# B&R Automation Studio project lab1_MIRTS_save2_4 (part 2)

```iecst
TYPE
    ARNC0FILEMONENTRY_typ : STRUCT
        name                            : UDINT;                                 (* File name (address) *)
        path_name                       : UDINT;                                 (* Full path file name (address) *)
        dir_name                        : UDINT;                                 (* Directory name (address) *)
        device_name                     : UDINT;                                 (* Device name (address) *)
        prog_nr                         : UDINT;                                 (* Number of loaded program *)
        storage_type                    : UDINT;                                 (* Storage type: 1-file, 2-module *)
        time_stamp                      : UDINT;                                 (* File time stamp *)
        precompiled_lcf                 : BOOL;                                  (* Loaded file is laguage configuration file *)
        NOT_USE_1                       : ARRAY[0..2] OF USINT;
        next                            : UDINT;                                 (* Next element in file list *)
    END_STRUCT;
    ARNC0FILEMONBASIC_typ : STRUCT
        name                            : STRING[31];                            (* Name of loaded file *)
        prog_nr                         : UDINT;                                 (* Number of loaded program *)
        storage_type                    : UDINT;                                 (* Storage type: 1-file, 2-module *)
    END_STRUCT;
    ARNC0FILEMONACCESS_typ : STRUCT
        valid                           : BOOL;                                  (* Extended data can be accessed *)
        NOT_USE_1                       : ARRAY[0..2] OF USINT;
        first                           : UDINT;                                 (* Begin of the file list *)
    END_STRUCT;
    ARNC0FILEMON_typ : STRUCT
        set_offset                      : UDINT;                                 (* Required file offset *)
        offset                          : UDINT;                                 (* Offset of displayed files *)
        file                            : ARRAY[0..31] OF ARNC0FILEMONBASIC_typ; (* File monitor *)
        direct_access                   : ARNC0FILEMONACCESS_typ;                (* Access to extended data *)
        handshake                       : BOOL;                                  (* Set to update data *)
        NOT_USE_1                       : ARRAY[0..2] OF USINT;
    END_STRUCT;
    ARNC0EXTWMCOL_typ : STRUCT
        result                          : UDINT;                                 (* WM result *)
        index1                          : UDINT;                                 (* Index of 1st found colliding area *)
        shape1                          : UDINT;                                 (* Shape of colliding area: 1-block, 2-hspace *)
    END_STRUCT;
    ARNC0EXTWM_typ : STRUCT
        joint_position                  : ARRAY[0..11] OF LREAL;                 (* Joint coordinate *)
        xyz_position                    : ARRAY[0..2] OF LREAL;                  (* TCP position if joints cannot be used *)
        D_FULL                          : ARRAY[0..5] OF LREAL;                  (* General tool *)
        local_frame                     : ARRAY[0..5] OF LREAL;                  (* Local (base) frame *)
        collision                       : ARNC0EXTWMCOL_typ;                     (* Additional information about collisions *)
    END_STRUCT;
    OPTMOT_SEG_CONFIG_typ : STRUCT
        distance                        : LREAL;                                 (* Length of the path segments in CNC units *)
        increase_num_seg_from_radius    : LREAL;                                 (* Finer segmentation of circles with smaller radius *)
        increase_num_seg_orient_factor  : LREAL;                                 (* Finer segmentation of orientation change *)
        G126_num_seg                    : UDINT;                                 (* Finer segmentation of rounding edge *)
        G126_num_seg_PTP_Interp         : UDINT;                                 (* Finer segmentation of rounding edge *)
    END_STRUCT;
    OPTMOT_AXES_typ : STRUCT
        ax_count                        : UDINT;                                 (* Number of axes for optimization *)
        ax_index                        : ARRAY [0..14] OF USINT;                (* Index of CNC-axis *)
        NOT_USE_1                       : USINT;
        ax_factor                       : ARRAY [0..14] OF LREAL;                (* Scaling factor *)
    END_STRUCT;
    OPTMOT_PATHDEF_typ : STRUCT
        type                            : UINT;                                  (* Type of path definition *)
        ax_count                        : UINT;                                  (* Number of axes for path computation *)
        ax_index                        : ARRAY [0..14] OF USINT;                (* Index of CNC-axis *)
        NOT_USE_1                       : USINT;
        ax_factor                       : ARRAY [0..14] OF LREAL;                (* Scaling factor *)
    END_STRUCT;
    OPTMOT_TRF_VAR_INSTANCES_typ : STRUCT
        trf_var_ip                      : UDINT;                                 (* For developers only *)
        trf_var_ip_wm                   : UDINT;                                 (* For developers only *)
        trf_var_pp1                     : UDINT;                                 (* For developers only *)
        trf_var_pp2                     : UDINT;                                 (* For developers only *)
        trf_var_bgen                    : UDINT;                                 (* For developers only *)
    END_STRUCT;
    OPTMOT_ACCESS_POINTS_typ : STRUCT
        pp_context                      : UDINT;                                 (* Access of data for external workspace monitoring *)
        wm_function                     : UDINT;                                 (* Access for external call of workspace monitoring *)
        address_debug_data              : UDINT;                                 (* For developers only *)
        trf_var_instances               : OPTMOT_TRF_VAR_INSTANCES_typ;          (* Structure of access points for developers only *)
    END_STRUCT;
    OPTMOT_INTERNAL_typ : STRUCT
        buffer_nc_block                 : UDINT;                                 (* Size of a buffer containing NC-blocks *)
        buffer_geometric_data           : UDINT;                                 (* Size of a buffer containing geometric data of the path *)
        disable_optmot_for_channel      : USINT;                                 (* Deactivation of optimizer for current CNC channel *)
        Ts_multiple                     : USINT;                                 (* Sample time of trajectory planer *)
        linear_feed                     : USINT;                                 (* Behavior of path acceleration *)
        bypass_optmot                   : USINT;                                 (* Simulation mode *)
        addr_dyn_model                  : UDINT;                                 (* Pointer to the dynamic model *)
        der_num_poly_points             : UINT;                                  (* Number of segments used for derivatives computation *)
        geometric_pos_filter            : UINT;                                  (* Number of segments used for position filter *)
        buffer_level_lookahead          : UINT;                                  (* Minimal fill level of lookahead buffer *)
        G220_reduce_to_max_in_buffer    : UINT;                                  (* Reduction of G220 time *)
        sigma_diff_compute              : LREAL;                                 (* Lookahead of segmentation *)
        max_angle                       : LREAL;                                 (* Angle to detect stops on path *)
        access_points                   : OPTMOT_ACCESS_POINTS_typ;              (* Structure of access points for developers only *)
        reserve1                        : ARRAY [0..9] OF LREAL;                 (* For developers only *)
        reserve2                        : ARRAY [0..9] OF DINT;                  (* For developers only *)
    END_STRUCT;
    OPTMOT_LIMITS_typ : STRUCT
        v_joint_min                     : ARRAY [0..14] OF LREAL;                (* Minimal velocity limits of the joint axes *)
        v_joint_max                     : ARRAY [0..14] OF LREAL;                (* Maximal velocity limits of the joint axes *)
        a_joint_min                     : ARRAY [0..14] OF LREAL;                (* Minimal acceleration limits of the joint axes *)
        a_joint_max                     : ARRAY [0..14] OF LREAL;                (* Maximal acceleration limits of the joint axes *)
        j_joint_min                     : ARRAY [0..14] OF LREAL;                (* Minimal jerk limits of the joint axes *)
        j_joint_max                     : ARRAY [0..14] OF LREAL;                (* Maximal jerk limits of the joint axes *)
        torque_min                      : ARRAY [0..14] OF LREAL;                (* Minimal torque limits of the joint axes *)
        torque_max                      : ARRAY [0..14] OF LREAL;                (* Maximal torque limits of the joint axes *)
        torque_limits_in_generator_mode : UDINT;                                 (* Activation of generator mode *)
        torque_gen_factor_min           : ARRAY [0..14] OF LREAL;                (* Factor for minimal torque limit in generator mode *)
        torque_gen_factor_max           : ARRAY [0..14] OF LREAL;                (* Factor for maximal torque limit in generator mode *)
        v_path_min                      : ARRAY [0..31] OF LREAL;                (* Minimal velocity limits of the path definitions *)
        v_path_max                      : ARRAY [0..31] OF LREAL;                (* Maximal velocity limits of the path definitions *)
        a_path_min                      : ARRAY [0..31] OF LREAL;                (* Minimal acceleration limits of the path definitions *)
        a_path_max                      : ARRAY [0..31] OF LREAL;                (* Maximal acceleration limits of the path definitions *)
        j_path_min                      : ARRAY [0..31] OF LREAL;                (* Minimal jerk limits of the path definitions *)
        j_path_max                      : ARRAY [0..31] OF LREAL;                (* Maximal jerk limits of the path definitions *)
    END_STRUCT;
    OPTMOT_ACTIVE_LIMIT_typ : STRUCT
        type                            : USINT;                                 (* Type of the active limit *)
        source                          : USINT;                                 (* Source of the active limit *)
        min_max                         : SINT;                                  (* Positive or negative range of the active limit *)
        index                           : USINT;                                 (* Index of the axis or path definition of the active limit *)
    END_STRUCT;
    OPTMOT_UNFILTERED_MONITOR_typ : STRUCT
        s_joint                         : ARRAY [0..14] OF LREAL;                (* Cyclical joint position in CNC units *)
        v_joint                         : ARRAY [0..14] OF LREAL;                (* Cyclical joint velocity in CNC units *)
        a_joint                         : ARRAY [0..14] OF LREAL;                (* Cyclical joint acceleration in CNC units *)
        j_joint                         : ARRAY [0..14] OF LREAL;                (* Cyclical joint jerk in CNC units *)
    END_STRUCT;
    OPTMOT_MONITOR_typ : STRUCT
        s_joint                         : ARRAY [0..14] OF LREAL;                (* Cyclical joint position in CNC units *)
        v_joint                         : ARRAY [0..14] OF LREAL;                (* Cyclical joint velocity in CNC units *)
        a_joint                         : ARRAY [0..14] OF LREAL;                (* Cyclical joint acceleration in CNC units *)
        j_joint                         : ARRAY [0..14] OF LREAL;                (* Cyclical joint jerk in CNC units *)
        feed_forward_torque             : ARRAY [0..14] OF LREAL;                (* Cyclical joint torque/force *)
        v_path                          : ARRAY [0..31] OF LREAL;                (* Cyclical path velocity in CNC units *)
        unfiltered_monitor              : OPTMOT_UNFILTERED_MONITOR_typ;         (* Monitor data without filters and override *)
        active_limit                    : OPTMOT_ACTIVE_LIMIT_typ;               (* Structure of information about current limitation *)
        data_valid                      : UINT;                                  (* Feed forward data is valid *)
        fill_level_lookahead            : UINT;                                  (* Fill level of lookahead buffer *)
        reserve                         : ARRAY [0..1] OF UDINT;
    END_STRUCT;
    OPTMOT_COND_STOP_typ : STRUCT
        active                          : UINT;                                  (* Conditional stop active *)
        call_stop_internal              : UINT;                                  (* Internal execution of the conditional stop *)
        identifier                      : UDINT;                                 (* Identifier of the conditional stop *)
        select_overlapped_identifier    : UDINT;                                 (* Selection of identifier in overlapping conditional stops *)
        select_identifier_stop_internal : UDINT;                                 (* Selection of identifier if conditional stop is executed internally *)
    END_STRUCT;
    OPTMOT_COND_STOP_OPTMOT_typ : STRUCT
        identifier_aktiv                : UDINT;                                 (* Output of aktive identifier *)
        identifier_fulfilled            : UDINT;                                 (* Input of fulfilled identifier *)
    END_STRUCT;
    OPTMOT_STOPPING_typ : STRUCT
        G126_skip_if_stop               : UINT;                                  (* Skip G126 if a stop on path occurs *)
        trajectory                      : UINT;                                  (* Definition of stopping trajectory *)
        conditional_stop                : OPTMOT_COND_STOP_typ;                  (* Structure of conditional stop *)
        conditional_stop_optmot         : OPTMOT_COND_STOP_OPTMOT_typ;           (* Structure of optmot synchronal conditional stop *)
    END_STRUCT;
    OPTMOT_PATH_typ : STRUCT
        G126_skip_smaller_radius        : LREAL;                                 (* Skip G126 if programmed radius is smaller *)
        G126_round_whole_line           : UDINT;                                 (* Round whole first/last line *)
        count                           : UDINT;                                 (* Number of path definitions *)
        definition                      : ARRAY [0..31] OF OPTMOT_PATHDEF_typ;   (* Structure of path definitions parameters *)
        stopping                        : OPTMOT_STOPPING_typ;                   (* Structure of stopping parameters *)
        reserve1                        : ARRAY [0..170] OF UDINT;
    END_STRUCT;
    OPTMOT_CONFIG_typ : STRUCT
        axes                            : OPTMOT_AXES_typ;                       (* Structure of joint axes parameters *)
        path                            : OPTMOT_PATH_typ;                       (* Structure of path parameters *)
        limits                          : ARRAY [0..31] OF OPTMOT_LIMITS_typ;    (* Structure of limit parameters *)
        segmentation                    : OPTMOT_SEG_CONFIG_typ;                 (* Structure of segmentation parameters *)
        monitor                         : OPTMOT_MONITOR_typ;                    (* Structure of monitor parameters *)
        internals                       : OPTMOT_INTERNAL_typ;                   (* Structure of internal parameters *)
    END_STRUCT;
    OPTMOT_MONITOR_ADVANCED_typ : STRUCT
        s_joint                         : ARRAY [0..14] OF LREAL;                (* Cyclical joint position in CNC units *)
        v_joint                         : ARRAY [0..14] OF LREAL;                (* Cyclical joint velocity in CNC units *)
        a_joint                         : ARRAY [0..14] OF LREAL;                (* Cyclical joint acceleration in CNC units *)
        j_joint                         : ARRAY [0..14] OF LREAL;                (* Cyclical joint jerk in CNC units *)
        feed_forward_torque             : ARRAY [0..14] OF LREAL;                (* Cyclical joint torque/force *)
        v_path                          : ARRAY [0..31] OF LREAL;                (* Cyclical path velocity in CNC units *)
        unfiltered_monitor              : OPTMOT_UNFILTERED_MONITOR_typ;         (* Monitor data without filters and override *)
        active_limit                    : OPTMOT_ACTIVE_LIMIT_typ;               (* Structure of information about current limitation *)
        data_valid                      : UINT;                                  (* Feed forward data is valid *)
        fill_level_lookahead            : UINT;                                  (* Fill level of lookahead buffer *)
        tracking_active                 : UINT;                                  (* Tracking active *)
        tracking_synch                  : UINT;                                  (* Robot synchronized with conveyor *)
        tracking_index                  : UINT;                                  (* Active tracking index *)
        reserve                         : UINT;
    END_STRUCT;
    OPTMOT_TRACKING_ORIENTATION_typ : STRUCT
        phi                             : LREAL;                                 (* Phi-component of a rotation *)
        theta                           : LREAL;                                 (* Theta-component of a rotation *)
        psi                             : LREAL;                                 (* Psi-component of a rotation *)
    END_STRUCT;
    OPTMOT_TRACKING_ORIENT_PARAM_typ : STRUCT
        measure                         : UDINT;                                 (* Unit of measurement of the angles *)
        angles_type                     : UDINT;                                 (* Angles type *)
    END_STRUCT;
    OPTMOT_TRACKING_LIMITS_typ : STRUCT
        maxVelocity                     : LREAL;                                 (* Maximal velocity of the conveyor belt *)
    END_STRUCT;
    OPTMOT_TRACKING_CYCLIC_typ : STRUCT
        position                        : LREAL;                                 (* Cyclical position of the conveyor belt *)
        velocity                        : LREAL;                                 (* Cyclical velocity of the conveyor belt *)
    END_STRUCT;
    OPTMOT_TRACKING_CONVEYOR_typ : STRUCT
        limits                          : OPTMOT_TRACKING_LIMITS_typ;            (* Structure of conveyor limits *)
        orientation                     : OPTMOT_TRACKING_ORIENTATION_typ;       (* Structure of orientation between global basic frame and conveyor belt frame *)
        cyclicData                      : OPTMOT_TRACKING_CYCLIC_typ;            (* Structure of cyclic data *)
    END_STRUCT;
    OPTMOT_TRACKING_CONVEYORDATA_typ : STRUCT
        orientationParameter            : OPTMOT_TRACKING_ORIENT_PARAM_typ;      (* Structure of general orientation parameters *)
        conveyor                        : ARRAY [0..9] OF OPTMOT_TRACKING_CONVEYOR_typ; (* Structure of conveyor belt data *)
    END_STRUCT;
    OPTMOT_TRACKING_typ : STRUCT
        enable                          : UDINT;                                 (* Enable tracking *)
        conveyorData                    : OPTMOT_TRACKING_CONVEYORDATA_typ;      (* Structure of conveyor belt tracking *)
        reserve1                        : ARRAY [0..7] OF LREAL;                 (* For developers only *)
        reserve2                        : ARRAY [0..31] OF UDINT;                (* For developers only *)
    END_STRUCT;
    OPTMOT_PATH_ADVANCED_typ : STRUCT
        G126_skip_smaller_radius        : LREAL;                                 (* Skip G126 if programmed radius is smaller *)
        G126_round_whole_line           : UDINT;                                 (* Round whole first/last line *)
        count                           : UDINT;                                 (* Number of path definitions *)
        definition                      : ARRAY [0..31] OF OPTMOT_PATHDEF_typ;   (* Structure of path definitions parameters *)
        stopping                        : OPTMOT_STOPPING_typ;                   (* Structure of stopping parameters *)
        tracking                        : OPTMOT_TRACKING_typ;                   (* Structure of tracking parameters *)
    END_STRUCT;
    OPTMOT_CONFIG_ADVANCED_typ : STRUCT
        axes                            : OPTMOT_AXES_typ;                       (* Structure of joint axes parameters *)
        path                            : OPTMOT_PATH_ADVANCED_typ;              (* Structure of path parameters *)
        limits                          : ARRAY [0..31] OF OPTMOT_LIMITS_typ;    (* Structure of limit parameters *)
        segmentation                    : OPTMOT_SEG_CONFIG_typ;                 (* Structure of segmentation parameters *)
        monitor                         : OPTMOT_MONITOR_ADVANCED_typ;           (* Structure of monitor parameters *)
        internals                       : OPTMOT_INTERNAL_typ;                   (* Structure of internal parameters *)
    END_STRUCT;
    ARNC0PLOTDATA01_typ : STRUCT
        block_ncprog                    : UDINT;                       			 (* Block number *)
        line_ncprog                     : UDINT;                       			 (* Line number *)
        MpId                            : UDINT;                       			 (* Motion packet ident *)
        MpSubId                         : UDINT;                       			 (* Motion packet subident *)
        cmd_code                        : UINT;                       			 (* Command *)
        reserve                         : UINT;                       			 (* don't use *)
        data                            : ARRAY [0..51] OF USINT;                (* Data *)
    END_STRUCT;
    ARNC0PLOTDATA02_typ : STRUCT
        block_ncprog                    : UDINT;                       			 (* Block number *)
        line_ncprog                     : UDINT;                       			 (* Line number *)
        MpId                            : UDINT;                       			 (* Motion packet ident *)
        MpSubId                         : UDINT;                       			 (* Motion packet subident *)
        cmd_code                        : UINT;                       			 (* Command *)
        reserve                         : UINT;                       			 (* don't use *)
        data                            : ARRAY [0..51] OF USINT;                (* Data *)
    END_STRUCT;
    ARNC0PLDMOVE_typ : STRUCT
        ep                              : ARRAY [0..2] OF REAL;                  (* End point *)
        cp                              : ARRAY [0..2] OF REAL;                  (* Center point *)
        radius                          : REAL;                                  (* Tool radius *)
        v_ncprog                        : REAL;                                  (* Programmed feedrate *)
        info                            : UDINT;                                 (* Info bits *)
    END_STRUCT;
    ARNC0PLDMOVE02_typ : STRUCT
        ep                              : ARRAY [0..2] OF REAL;                  (* End point *)
        cp                              : ARRAY [0..2] OF REAL;                  (* Center point *)
        radius                          : REAL;                                  (* Tool radius *)
        v_ncprog                        : REAL;                                  (* Programmed feedrate *)
        t                               : REAL;                                  (* block runtime *)
        s                               : REAL;                                  (* block length, interpolated axes *)
        s_all                           : REAL;                                  (* block length, all axes *)
        info                            : UDINT;                                 (* Info bits *)
    END_STRUCT;
    ARNC0PLDPROGEND_typ : STRUCT
        t                               : REAL;                                  (* estimated runtime *)
        s                               : REAL;                                  (* path length, interpolated axes *)
        s_all                           : REAL;                                  (* path length, all axes *)
    END_STRUCT;
    ARNC0PLDPROGSTART_typ : STRUCT
        ProgNumber                      : UDINT;                                 (* program number *)
    END_STRUCT;
    ARNC0PLDTOOL_typ : STRUCT
        radius                          : REAL;                                  (* Tool radius *)
        length                          : REAL;                                  (* Tool length *)
        offset                          : ARRAY [0..2] OF REAL;                  (* Tool offset *)
        index                           : UINT;                                  (* Tool index, tool data number *)
        reserve                         : UINT;                                  (* don't use *)
    END_STRUCT;
    ARNC0PLDCSTRF_typ : STRUCT
        matrix                          : ARRAY [0..8] OF REAL;                  (* Rotation matrix *)
        offset                          : ARRAY [0..2] OF REAL;                  (* Offset (cs + tool) *)
        info                            : UDINT;                                 (* Info bits *)
    END_STRUCT;
    ARNC0PLDUSER_typ : STRUCT
        data                            : ARRAY [0..51] OF USINT;                (* User data *)
    END_STRUCT;
    ARNC0TRFIODATA_typ : STRUCT
        status                          : UDINT;                                 (* Return status of the last call of the transformation function *)
        in_pos                          : ARRAY [0..11] OF LREAL;                (* Input positions of the transformation function *)
        in_pos_ext                      : ARRAY [0..11] OF LREAL;                (* Extended input positions of the transformation function *)
        out_pos                         : ARRAY [0..71] OF LREAL;                (* Output positions of the transformation function *)
        info                            : ARRAY [0..8] OF UDINT;                 (* Information about the last call of the transformation function *)
    END_STRUCT;
    ARNC0WSCTRL_typ : STRUCT
        link_index                      : UDINT;                                 (* index of colliding link *)
        link2_index                     : UDINT;                                 (* index of colliding link for self-collision *)
        area_index                      : UDINT;                                 (* index of colliding area *)
    END_STRUCT;
    ARNC0NCMON_EXT_AX_typ : STRUCT
        nc_object                       : UDINT;
        nc_object_plcopen               : UDINT;
        v                               : REAL;                                  (* axis limit [cnc unit/s] *)
        a                               : REAL;                                  (* axis limit [cnc unit/s2] *)
        t_jolt                          : REAL;                                  (* axis jolt filter [s] (cnc system) *)
        pos_sw_end                      : DINT;                                  (* [cnc unit] *)
        neg_sw_end                      : DINT;                                  (* [cnc unit] *)
        unitfactor                      : REAL;                                  (* cnc unit factor *)
        plcopen_factor                  : REAL;                                  (* PLCopen unit factor *)
        type                            : UDINT;                                 (* axis type *)
        rot_period                      : REAL;                                  (* period of the rotary axis [cnc unit] *)
        rot_offset                      : REAL;                                  (* period start offsetof the rotary axis [cnc unit] *)
        ipl_mode                        : USINT;                                 (* interpolation mode *)
        drive_axfilter                  : USINT;                                 (* axis jolt filter on drive enable/disable *)
        nc_obj_name                     : ARRAY [0..13] OF USINT;
        cnc_ax_name                     : ARRAY [0..13] OF USINT;
        reserve                         : ARRAY [0..1] OF USINT;
    END_STRUCT;
    ARNC0NCMON_EXT_G113_typ : STRUCT
        k_alpha_max                     : REAL;                                  (* G113 parameter *)
        alpha_min                       : REAL;                                  (* G113 parameter *)
        alpha_max                       : REAL;                                  (* G113 parameter *)
    END_STRUCT;
    ARNC0NCMON_EXT_CNC_typ : STRUCT
        nc_object                       : UDINT;                                 (* nc object (cnc) *)
        v                               : REAL;                                  (* path limit [cnc unit/s] *)
        a_pos                           : REAL;                                  (* path limit [cnc unit/s2] *)
        a_neg                           : REAL;                                  (* path limit [cnc unit/s] *)
        t_jolt                          : REAL;                                  (* path jolt filter [s] *)
        feed                            : REAL;                                  (* programmed feed [cnc unit/s] *)
        v_jump                          : ARRAY [0..14] OF REAL;                 (* speed jump [cnc unit/s] *)
        a_jump                          : ARRAY [0..14] OF REAL;                 (* acceleration jump [cnc unit/s] *)
        v_jump_t                        : REAL;                                  (* speed jump for tangential axes [cnc unit/s] *)
        s_jump_t                        : REAL;                                  (* blocktransition tangential / non tangential [deg] *)
        filter_err_cir                  : REAL;                                  (* allowed radius error (jolt filter) [cnc unit] *)
        filter_err_trans                : REAL;                                  (* contour violation (jolt filter) [cnc unit] *)
        radius_err                      : REAL;                                  (* center point prgramming [cnc unit] *)
        elements                        : UDINT;                                 (* calculated elements before start *)
        block_buffer                    : UDINT;                                 (* block buffer for backtracing *)
        lookahead                       : UDINT;                                 (* look ahead buffer (dynamics calculation) *)
        first_M                         : UINT;                                  (* index of 1st M function (without sync) *)
        last_M                          : UINT;                                  (* index of last M function (without sync) *)
        first_M_S                       : UINT;                                  (* index of 1st M function (with sync) *)
        last_M_S                        : UINT;                                  (* index of last M function (with sync) *)
        s_sync1_t                       : UINT;                                  (* 1st sync M function (G141) *)
        s_sync2_t                       : UINT;                                  (* 2nd sync M function (G141) *)
        blocktransition                 : USINT;                                 (* block transition mode *)
        reserve                         : USINT;
        nc_obj_name                     : ARRAY [0..13] OF USINT;
        g113_data                       : ARNC0NCMON_EXT_G113_typ;
    END_STRUCT;
    ARNC0NCMON_EXT_G705_typ : STRUCT
        ident                           : UDINT;                                 (* G705 ident *)
        axis                            : ARRAY[0..14] OF ARNC0NCMON_EXT_AX_typ;
        cnc                             : ARNC0NCMON_EXT_CNC_typ;
        block_ncprog                    : UDINT;                                 (* block number (G705) *)
        line_ncprog                     : UDINT;                                 (* line number (G705) *)
        cnc_channel                     : UINT;                                  (* cnc channel (idndex) *)
        reserve                         : UINT;
    END_STRUCT;
    ARNC0NCMON_EXT_typ : STRUCT
        s_set                           : ARRAY [0..14] OF LREAL;                (* set position *)
        s_ncprog                        : LREAL;                                 (* path position in current CNC program *)
        g705_data                       : ARNC0NCMON_EXT_G705_typ;               (* parameter at program start, at G705 *)
        reserve                         : ARRAY[0..1] OF UDINT;
    END_STRUCT;
    ARNC0WFM_SERIAL_typ : STRUCT
        nr_of_points : UDINT;                                                    (* number of points of wire-frame model *)
        point : ARRAY[0..20, 0..2] OF LREAL;                                     (* points of wire-frame model *)
        nr_of_arms : UDINT;                                                      (* number of arm diameters *)
        arm_diameter : ARRAY[0..19] OF LREAL;                                    (* arm diameters *)
        safe_distance : LREAL;                                                   (* safe distance *)
    END_STRUCT;
    ARNC0WFM_COMPLETE_typ : STRUCT
        data : ARRAY[0..329] OF UDINT;                                           (* internal data of complete wire-frame model *)
    END_STRUCT;
    ARNC0WFM_typ : STRUCT
        use_complete : UDINT;                                                    (* use complete type of wire-frame model *)
        complete : ARNC0WFM_COMPLETE_typ;                                        (* complete wire-frame model data *)
        use_serial : UDINT;                                                      (* use serial type of wire-frame model *)
        serial : ARNC0WFM_SERIAL_typ;                                            (* serial wire-frame model data *)
    END_STRUCT;
    ARNC0WFM_BFS : STRUCT
        enable : UDINT;                                                          (* enable frame *)
        dx : LREAL;                                                              (* x transition *)
        dy : LREAL;                                                              (* y transition *)
        dz : LREAL;                                                              (* z transition *)
        phi : LREAL;                                                             (* angle in meaning of angles type *)
        theta : LREAL;                                                           (* angle in meaning of angles type *)
        psi : LREAL;                                                             (* angle in meaning of angles type *)
        angles_type : UDINT;                                                     (* angles type *)
    END_STRUCT;
    ARNC0WFM_MON_typ : STRUCT
        valid_data : UDINT;                                                      (* number of calls with valid data *)
        invalid_data : UDINT;                                                    (* number of calls with invalid data *)
    END_STRUCT;
    ARNC0WFM_EXT_typ : STRUCT
        p_wire_frame_model : REFERENCE TO ARNC0WFM_typ;                          (* reference to wire-frame model data *)
        base_frame_shift : ARNC0WFM_BFS;                                         (* frame *)
        monitor : ARNC0WFM_MON_typ;                                              (* monitor *)
    END_STRUCT;
    ARNC0INTERACTION_typ : STRUCT
        wire_frame_model : ARNC0WFM_typ;                                         (* wire-frame model data *)
        wire_frame_models_to_check : ARRAY[0..23]OF ARNC0WFM_EXT_typ;            (* array of wire-frame models data *)
    END_STRUCT;
END_TYPE
TYPE
  ARNC0IP_MON_typ : STRUCT
    enable : USINT;                             (*Enable cyclic update *)
    reserve : ARRAY[0..2] OF USINT;             (*[RESERVE] *)
    status_msg : ARRAY[0..79] OF USINT;         (*String: current status of interpreter e.g. Running/Waiting/Finished *)
    last_error_msg : ARRAY[0..119] OF USINT;    (*String: last error message issued *)
    last_error_code : UINT ;                    (*Last status message code issued *)
    loaded_prog_count : UINT ;                  (*Number of files loaded *)
    prog_name : ARRAY[0..79] OF USINT;          (*Name of start-program *)
    ncblock_l2 : ARRAY[0..79] OF USINT;         (*Interpeter block monitor: current line -2 *)
    ncblock_l1 : ARRAY[0..79] OF USINT;         (*Interpeter block monitor: current line -1 *)
    ncblock : ARRAY[0..79] OF USINT;            (*Interpeter block monitor: current line *)
    ncblock_n1 : ARRAY[0..79] OF USINT;         (*Interpeter block monitor: current line +1 *)
    ncblock_n2 : ARRAY[0..79] OF USINT;         (*Interpeter block monitor: current line +2 *)
    cur_line_num : UDINT ;                      (*Interpeter block monitor: current line number *)
    cur_block_num : UDINT ;                     (*Interpeter block monitor: current line N-block number *)
    intern1 : UDINT ;                           (*[INTERNAL] *)
    intern2 : UDINT ;                           (*[INTERNAL] *)
    intern3 : UDINT ;                           (*[INTERNAL] *)
    intern4 : UDINT ;                           (*[INTERNAL] *)
    intern5 : UDINT ;                           (*[INTERNAL] *)
    breakpoint_count : UDINT ;                  (*Number of breakpoints set *)
    ipvar_access_count : UDINT ;                (*Number of IP variables being directly accessed by PLC *)
    intern6 : UDINT ;                           (*[INTERNAL] *)
    intern7 : UDINT ;                           (*[INTERNAL] *)
    num_parallel_events : UDINT ;               (*Number of cyclic jobs currently active *)
    parallel_cycle_count : UDINT ;              (*Number of execution cycles of all cyclic jobs *)
    parallel_action_text : ARRAY[0..11, 0..79] OF USINT; (*cyclic execution monitor - cyclic job source line text *)
    parallel_eval_count : ARRAY[0..11] OF UDINT ;   (*number of times the cyclic job has been evaluated (tested) *)
    parallel_exec_count : ARRAY[0..11] OF UDINT ;   (*number of times a Synchronised Action has executed (not relevant to FUBs) *)
    num_fubs_exec_ipsynch : UDINT ;             (*Number of interpreter synchronous FUBs executing *)
    num_fubs_exec_ppsynch : UDINT ;             (*Number of path synchronous FUBs executing *)
    callstack : ARRAY[0..11, 0..79] OF USINT;   (*Program callstack *)
    shared_mem_size : UDINT ;                   (*Memory consumed by shared library data (partitions will be larger) *)
    ip_mem_size : UDINT ;                       (*Memory consumed by interpreter instance (partitions will be larger) *)
    ip_cur_file_mem_size : UDINT ;              (*Memory consumed by start program (or last loaded program) file (partitions will be larger) *)
    sys_free_mem : UDINT ;                      (*Available system memory *)
    intern8 : UDINT ;                           (*[INTERNAL] *)
    intern9 : UDINT ;                           (*[INTERNAL] *)
    intern10 : UDINT ;                          (*[INTERNAL] *)
    intern11 : UDINT ;                          (*[INTERNAL] *)
    parallel_enabled : USINT ;                  (*Bool: cyclic execution enabled *)
    parallel_rdisable_set : USINT ;             (*Bool: cyclic jobs set the keep-alive (rdisable) flag *)
    intern12 : USINT ;                          (*[INTERNAL] *)
    intern13 : USINT ;                          (*[INTERNAL] *)
    cur_prog_file_name : ARRAY[0..79] OF USINT ;(*File name of the current program*)
    cur_prog_name : ARRAY[0..79] OF USINT ;     (*Name of the current program*)
  END_STRUCT;
END_TYPE
```

- acp10err-en.txt (not shown)

- arnc0err-de.txt (not shown)

- arnc0err-en.txt (not shown)

### Library Logical/Libraries/MotorCntrl (ANSIC)

#### MotorCntrl.fun - Exported functions and function blocks
```iecst
{REDUND_ERROR} FUNCTION_BLOCK FB_Motor (*TODO: Add your comment here*) (*$GROUP=User,$CAT=User,$GROUPICON=User.png,$CATICON=User.png*)
	VAR_INPUT
		u : {REDUND_UNREPLICABLE} REAL; (*Входное напряжение [B]*)
	END_VAR
	VAR_OUTPUT
		w : REAL; (*Частота вращения [об/мин]*)
		phi : REAL; (*Положение [рад]*)
	END_VAR
	VAR
		integrator : FB_Integrator; (*Интегратор*)
		Tm : REAL; (*Электромеханическая постоянная времени [с]*)
		ke : REAL; (*Постоянная ЭДС двигателя [В*мин/об]*)
		dt : REAL; (*Шаг расчета [с]*)
	END_VAR
END_FUNCTION_BLOCK

{REDUND_ERROR} FUNCTION_BLOCK FB_Regulator (*TODO: Add your comment here*) (*$GROUP=User,$CAT=User,$GROUPICON=User.png,$CATICON=User.png*)
	VAR_INPUT
		e : {REDUND_UNREPLICABLE} REAL; (*Рассогласование между задающим воздействием и реальной скоростью вращения вала ДПТ [об/мин]*)
	END_VAR
	VAR_OUTPUT
		u : REAL; (*Напряжение, подаваемое на вход ДПТ [B]*)
	END_VAR
	VAR
		k_p : REAL; (*Пропорциональный коэффициент регулятора*)
		k_i : REAL; (*Интегральный коэффициент регулятора*)
		integrator : FB_Integrator; (*Интегратор*)
		ivOld : REAL; (*Хранение предыдущего значения схемы противонакопления*)
		max_abs_value : REAL; (*Граница блока ограничения [В]*)
		dt : REAL; (*Шаг расчета [c]*)
	END_VAR
END_FUNCTION_BLOCK

{REDUND_ERROR} FUNCTION_BLOCK FB_Integrator (*TODO: Add your comment here*) (*$GROUP=User,$CAT=User,$GROUPICON=User.png,$CATICON=User.png*)
	VAR_INPUT
		in : {REDUND_UNREPLICABLE} REAL; (*Вход интегрирующего звена*)
	END_VAR
	VAR_OUTPUT
		out : REAL; (*Выход интегрирующего звена*)
	END_VAR
	VAR
		dt : REAL; (*Шаг расчета [c]*)
	END_VAR
END_FUNCTION_BLOCK
```

#### FB_Motor.c
```c
#include <bur/plctypes.h>
#ifdef __cplusplus
	extern "C"
	{
#endif
#include "MotorCntrl.h"
#ifdef __cplusplus
	};
#endif
/* TODO: Add your comment here */
void FB_Motor(struct FB_Motor* inst)
{
	/*TODO: Add your code here*/
	inst->integrator.dt = inst->dt;
	inst->integrator.in = ((inst->u)/(inst->ke) - (inst->w))*\
		(1/(inst->Tm));
	FB_Integrator(&(inst->integrator));
	inst->w = inst->integrator.out;
	inst->integrator.in = inst->w;
	inst->integrator.out = inst->phi;
	FB_Integrator(&(inst->integrator));
	inst->phi = inst->integrator.out;
	inst->integrator.out = inst->w;
}
```

#### FB_Regulator.c
```c
#include <bur/plctypes.h>
#ifdef __cplusplus
	extern "C"
	{
#endif
#include "MotorCntrl.h"
#ifdef __cplusplus
	};
#endif
/* TODO: Add your comment here */
REAL V_lim(REAL in, REAL max_in)
{
	if ((in >= max_in) || (in <= -max_in))
	{
		if (in>0)
			return max_in;
		else
			return -max_in;
	}
	else
		return in;
}
void FB_Regulator(struct FB_Regulator* inst)
{
	/*TODO: Add your code here*/
	REAL temp;
	inst->integrator.dt = inst->dt;
	inst->integrator.in = ((inst->e*inst->k_i)+inst->ivOld);
	FB_Integrator(&(inst->integrator));
	temp = inst->integrator.out + V_lim((inst->e)*(inst->k_p),inst->max_abs_value);
	inst->u = V_lim(temp, inst->max_abs_value);
	inst->ivOld = inst->u - temp;
}
```

#### FB_Integrator.c
```c
#include <bur/plctypes.h>
#ifdef __cplusplus
	extern "C"
	{
#endif
#include "MotorCntrl.h"
#ifdef __cplusplus
	};
#endif
/* TODO: Add your comment here */
void FB_Integrator(struct FB_Integrator* inst)
{
	/*TODO: Add your code here*/
	inst->out += (inst->in)*(inst->dt);
}
```

### Program Logical/LedCtrl (ANSIC)

#### Main.c
```c
#include <bur/plctypes.h>

#ifdef _DEFAULT_INCLUDES
	#include <AsDefault.h>
#endif

void _INIT ProgramInit(void)
{

}

void _CYCLIC ProgramCyclic(void)
{
		sc0 = sw0;
		sc1 = sw1;
		sc2 = sw2;
		sc3 = sw3;

}

void _EXIT ProgramExit(void)
{

}
```

### Program Logical/ncsdcctrl

#### ncsdcctrl.var
```iecst
VAR
	gAxis01_oSetPosOld : INT := 0;
	gAxis02_oSetPosOld : INT := 0;
	gAxis04_oSetPosOld : INT := 0;
	gAxis05_oSetPosOld : INT := 0;
END_VAR
```

#### ncsdcctrlCyclic.st
```iecst
PROGRAM _CYCLIC

(* ### BEGIN gAxis01 ### *)

(* life counter emulation of digital inputs *)
      gAxis01_DiDoIf.iLifeCntReference := gAxis01_DiDoIf.iLifeCntReference + 1;
      gAxis01_DiDoIf.iLifeCntNegHwEnd  := gAxis01_DiDoIf.iLifeCntNegHwEnd  + 1;
      gAxis01_DiDoIf.iLifeCntPosHwEnd  := gAxis01_DiDoIf.iLifeCntPosHwEnd  + 1;

(* default function model of ACOPOSmicro: convert absolute steps to delta steps - overflow save delta calculation *)
      gAxis01_MotorStep0 := gAxis01_DrvIf.oSetPos - gAxis01_oSetPosOld;
      gAxis01_oSetPosOld := gAxis01_DrvIf.oSetPos;

(* ### END gAxis01 ### *)

(* ### BEGIN gAxis02 ### *)

(* life counter emulation of digital inputs *)
      gAxis02_DiDoIf.iLifeCntReference := gAxis02_DiDoIf.iLifeCntReference + 1;
      gAxis02_DiDoIf.iLifeCntNegHwEnd  := gAxis02_DiDoIf.iLifeCntNegHwEnd  + 1;
      gAxis02_DiDoIf.iLifeCntPosHwEnd  := gAxis02_DiDoIf.iLifeCntPosHwEnd  + 1;

(* default function model of ACOPOSmicro: convert absolute steps to delta steps - overflow save delta calculation *)
      gAxis02_MotorStep0 := gAxis02_DrvIf.oSetPos - gAxis02_oSetPosOld;
      gAxis02_oSetPosOld := gAxis02_DrvIf.oSetPos;

(* ### END gAxis02 ### *)

(* ### BEGIN gAxis03 ### *)

(* life counter emulation of digital inputs *)
        gAxis03_DiDoIf.iLifeCntReference := gAxis03_DiDoIf.iLifeCntReference + 1;
        gAxis03_DiDoIf.iLifeCntNegHwEnd  := gAxis03_DiDoIf.iLifeCntNegHwEnd  + 1;
        gAxis03_DiDoIf.iLifeCntPosHwEnd  := gAxis03_DiDoIf.iLifeCntPosHwEnd  + 1;

(* ### END gAxis03 ### *)

(* ### BEGIN gAxis04 ### *)

(* life counter emulation of digital inputs *)
      gAxis04_DiDoIf.iLifeCntReference := gAxis04_DiDoIf.iLifeCntReference + 1;
      gAxis04_DiDoIf.iLifeCntNegHwEnd  := gAxis04_DiDoIf.iLifeCntNegHwEnd  + 1;
      gAxis04_DiDoIf.iLifeCntPosHwEnd  := gAxis04_DiDoIf.iLifeCntPosHwEnd  + 1;

(* default function model of ACOPOSmicro: convert absolute steps to delta steps - overflow save delta calculation *)
      gAxis04_MotorStep0 := gAxis04_DrvIf.oSetPos - gAxis04_oSetPosOld;
      gAxis04_oSetPosOld := gAxis04_DrvIf.oSetPos;

(* ### END gAxis04 ### *)

(* ### BEGIN gAxis05 ### *)

(* life counter emulation of digital inputs *)
      gAxis05_DiDoIf.iLifeCntReference := gAxis05_DiDoIf.iLifeCntReference + 1;
      gAxis05_DiDoIf.iLifeCntNegHwEnd  := gAxis05_DiDoIf.iLifeCntNegHwEnd  + 1;
      gAxis05_DiDoIf.iLifeCntPosHwEnd  := gAxis05_DiDoIf.iLifeCntPosHwEnd  + 1;

(* default function model of ACOPOSmicro: convert absolute steps to delta steps - overflow save delta calculation *)
      gAxis05_MotorStep0 := gAxis05_DrvIf.oSetPos - gAxis05_oSetPosOld;
      gAxis05_oSetPosOld := gAxis05_DrvIf.oSetPos;

(* ### END gAxis05 ### *)

END_PROGRAM
```

#### ncsdcctrlInit.st
```iecst
PROGRAM _INIT

(* ### BEGIN gAxis01 ### *)

(* initialize general interfaces *)
      gAxis01.size := gAxis01.size;
      gAxis01_HW.DrvIf_Typ := ncSDC_DRVSM16;
      brsstrcpy( ADR(gAxis01_HW.DrvIf_Name[0]), ADR('gAxis01_DrvIf') );
      gAxis01_HW.DiDoIf_Typ := ncSDC_DIDO;
      brsstrcpy( ADR(gAxis01_HW.DiDoIf_Name[0]), ADR('gAxis01_DiDoIf') );
      gAxis01_HW.EncIf1_Typ := ncSDC_ENC16;
      brsstrcpy( ADR(gAxis01_HW.EncIf1_Name[0]), ADR('gAxis01_EncIf1') );
      gAxis01_EncIf1.iLifeCnt := gAxis01_EncIf1.iLifeCnt;

(* initialize old-value for delta step calculation *)
      gAxis01_oSetPosOld := gAxis01_DrvIf.oSetPos;

(* ### END gAxis01 ### *)

(* ### BEGIN gAxis02 ### *)

(* initialize general interfaces *)
      gAxis02.size := gAxis02.size;
      gAxis02_HW.DrvIf_Typ := ncSDC_DRVSM16;
      brsstrcpy( ADR(gAxis02_HW.DrvIf_Name[0]), ADR('gAxis02_DrvIf') );
      gAxis02_HW.DiDoIf_Typ := ncSDC_DIDO;
      brsstrcpy( ADR(gAxis02_HW.DiDoIf_Name[0]), ADR('gAxis02_DiDoIf') );
      gAxis02_HW.EncIf1_Typ := ncSDC_ENC16;
      brsstrcpy( ADR(gAxis02_HW.EncIf1_Name[0]), ADR('gAxis02_EncIf1') );
      gAxis02_EncIf1.iLifeCnt := gAxis02_EncIf1.iLifeCnt;

(* initialize old-value for delta step calculation *)
      gAxis02_oSetPosOld := gAxis02_DrvIf.oSetPos;

(* ### END gAxis02 ### *)

(* ### BEGIN gAxis03 ### *)

(* initialize variables *)
        gAxis03_HW.DrvIf_Typ := ncSDC_DRVSERVO16;
        brsstrcpy(ADR(gAxis03_HW.DrvIf_Name[0]), ADR('gAxis03_DrvIf'));
        gAxis03_HW.DiDoIf_Typ := ncSDC_DIDO;
        brsstrcpy(ADR(gAxis03_HW.DiDoIf_Name[0]), ADR('gAxis03_DiDoIf'));

(* force variable offset generation *)
        gAxis03.size                      := gAxis03.size;
        gAxis03_DrvIf.iLifeCnt            := gAxis03_DrvIf.iLifeCnt;
        gAxis03_DiDoIf.iLifeCntDriveReady := gAxis03_DiDoIf.iLifeCntDriveReady;
        gAxis03_ModuleOk                  := gAxis03_ModuleOk;

(* assign your hardware inputs here*)

(*      gAxis03_DiDoIf.iPosHwEnd  := gAxis03_DiDoIf.iPosHwEnd;
        gAxis03_DiDoIf.iNegHwEnd  := gAxis03_DiDoIf.iNegHwEnd;
        gAxis03_DiDoIf.iReference := gAxis03_DiDoIf.iReference;
 *)

(* ### END gAxis03 ### *)

(* ### BEGIN gAxis04 ### *)

(* initialize general interfaces *)
      gAxis04.size := gAxis04.size;
      gAxis04_HW.DrvIf_Typ := ncSDC_DRVSM16;
      brsstrcpy( ADR(gAxis04_HW.DrvIf_Name[0]), ADR('gAxis04_DrvIf') );
      gAxis04_HW.DiDoIf_Typ := ncSDC_DIDO;
      brsstrcpy( ADR(gAxis04_HW.DiDoIf_Name[0]), ADR('gAxis04_DiDoIf') );
      gAxis04_HW.EncIf1_Typ := ncSDC_ENC16;
      brsstrcpy( ADR(gAxis04_HW.EncIf1_Name[0]), ADR('gAxis04_EncIf1') );
      gAxis04_EncIf1.iLifeCnt := gAxis04_EncIf1.iLifeCnt;

(* initialize old-value for delta step calculation *)
      gAxis04_oSetPosOld := gAxis04_DrvIf.oSetPos;

(* ### END gAxis04 ### *)

(* ### BEGIN gAxis05 ### *)

(* initialize general interfaces *)
      gAxis05.size := gAxis05.size;
      gAxis05_HW.DrvIf_Typ := ncSDC_DRVSM16;
      brsstrcpy( ADR(gAxis05_HW.DrvIf_Name[0]), ADR('gAxis05_DrvIf') );
      gAxis05_HW.DiDoIf_Typ := ncSDC_DIDO;
      brsstrcpy( ADR(gAxis05_HW.DiDoIf_Name[0]), ADR('gAxis05_DiDoIf') );
      gAxis05_HW.EncIf1_Typ := ncSDC_ENC16;
      brsstrcpy( ADR(gAxis05_HW.EncIf1_Name[0]), ADR('gAxis05_EncIf1') );
      gAxis05_EncIf1.iLifeCnt := gAxis05_EncIf1.iLifeCnt;

(* initialize old-value for delta step calculation *)
      gAxis05_oSetPosOld := gAxis05_DrvIf.oSetPos;

(* ### END gAxis05 ### *)

END_PROGRAM
```

### Program Logical/Program

#### Variables.var
```iecst
VAR
	Speed : REAL;
	fb_motor2 : FB_Motor;
	counter : REAL;
	fb_regulator : FB_Regulator;
	fb_motor : FB_Motor;
	Enable : BOOL; (*Флаг активации СУ*)
END_VAR
```

#### Main.c
```c
#include <bur/plctypes.h>

#ifdef _DEFAULT_INCLUDES
#include <AsDefault.h>
#endif

void _INIT ProgramInit(void)
{
	fb_regulator.k_p = 66.7;
	fb_regulator.k_i = 1666.7;
	fb_regulator.ivOld = 0;
	fb_regulator.max_abs_value = 4000;
	fb_regulator.dt = 0.002;
	fb_regulator.e = 0;
	fb_regulator.u = 0;

	fb_motor.Tm = 0.04;
	fb_motor.ke = 10;
	fb_motor.dt = 0.002;
	fb_motor.u = 0;
	fb_motor.w = 0;
	fb_motor.phi = 0;

	fb_motor2.Tm = 0.04;
	fb_motor2.ke = 10;
	fb_motor2.dt = 0.002;
	fb_motor2.u = 0;
	fb_motor2.w = 0;
	fb_motor2.phi = 0;

	counter = 0;
	Speed = 0;
	Enable = 1;
}

void _CYCLIC ProgramCyclic(void)
{
	counter+=1;
	Speed = (counter <= 200)?60:0;
	if (counter == 1000)
	{
		counter = 0;
	}
	if (Enable)
	{
		fb_regulator.e = Speed - fb_motor.w;
		FB_Regulator(&fb_regulator);
		fb_motor.u = fb_regulator.u;
		FB_Motor(&fb_motor);

		fb_motor2.u = Speed - fb_motor2.w;
		FB_Motor(&fb_motor2);
	}
}

void _EXIT ProgramExit(void)
{

}
```

Listed in the project but not available here: Logical/Global.typ, Logical/Libraries/X64Lib/X64Lib.typ, Logical/Libraries/X64Lib/FBX64Inverter.c, Logical/Libraries/X64Lib/X64Lib.fun, Logical/Libraries/MotorCntrl/Types.typ, Logical/Libraries/MotorCntrl/Constants.var, Logical/DoorCtrl
